// SIMATIC S7-200 project (STEP 7-Micro/WIN), CPU 224XP CN REL 02.01

ORGANIZATION_BLOCK MAIN:OB1
TITLE= 
// PROGRAM COMMENTS
// Press F1 for help and example program
//  
BEGIN
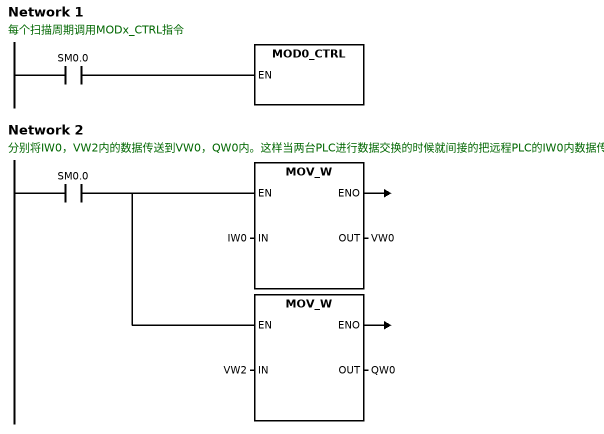
Network 1
// 每个扫描周期调用MODx_CTRL指令
LD     SM0.0
CALL   MOD0_CTRL:SBR1
Network 2
// 分别将IW0，VW2内的数据传送到VW0，QW0内。这样当两台PLC进行数据交换的时候就间接的把远程PLC的IW0内数据传送到本地PLC的QW0内，同时将本地PLC的IW0内的数据写入到远程PLC的QW0内
// (network saved uncompiled; LAD cells follow)
// row 0: c0 -| |- SM0.0 v  c1 --  c2 [MOV_W EN:=power@row0, IN:=IW0, ENO=>power, OUT=>VW0]  c3 ->
// row 1: c0 ^v  c2 [box]
// row 2: c0 ^  c1 --  c2 [MOV_W EN:=power@row2, IN:=VW2, ENO=>power, OUT=>QW0]  c3 ->
// row 3: c2 [box]
END_ORGANIZATION_BLOCK

// SBR1: protected block, not included

// (further data pages could not be read)
